INTERFACE ITrackList

METHOD FindMover : UDINT
VAR_INPUT
	status : INT;
END_VAR
END_METHOD

METHOD SetMoverInUse : BOOL;
VAR_INPUT
	moverNumber	: UDINT;
END_VAR
END_METHOD

METHOD SetMoverRef : BOOL
VAR_INPUT
	index : DINT;
	mover	: IMover;
END_VAR
END_METHOD

METHOD Sort : bool
VAR_INPUT
END_VAR
END_METHOD

METHOD UpdateMoverData : bool
VAR_INPUT
	data	: ST_MoverData;
END_VAR
END_METHOD

END_INTERFACE

(* stored: Version 1.1.0.1, ProductVersion 3.1.4026.12
   Itf ITrackList: Id {26cab804-596d-4864-8cd8-7d64b3c06639}
   Method FindMover: Id {1faee4eb-b871-41a3-a7e7-c273132636db}
   Method SetMoverInUse: Id {f099ce91-25b4-4f45-9d02-7efa3fb381ee}
   Method SetMoverRef: Id {f7d088c4-70d8-4371-b1e0-e360740f5625}
   Method Sort: Id {11abf748-dd65-48d2-bc1f-2500f31ada4d}
   Method UpdateMoverData: Id {2b01b911-4a74-4eee-a901-630b73283a40} *)
